// TwinCAT 3 PLC project Nepionic_PackML_Test
// ProgramVersion: 3.1.4026.21
// libraries:
//   [Nepionic_PackML], * (Nepionic)
//   Tc3_Module, * (Beckhoff Automation GmbH)
//   TcUnit, * (www.tcunit.org)
// project tree:
//   Mocks/ MockUnitMode.TcPOU
//   Programs/ TestRunner.TcPOU
//   Tasks/ TestRunnerTask.TcTTO
//   Tests/ PackMLTestSuite.TcPOU
// real-time tasks:
//   TASK TestRunnerTask: cycle T#10ms, priority 20, ADS port 350

CONFIGURATION Nepionic_PackML_Test
    RESOURCE PLC ON TwinCAT3
        TASK TestRunnerTask(INTERVAL := T#10ms, PRIORITY := 20);
        PROGRAM TestRunner WITH TestRunnerTask : TestRunner;
    END_RESOURCE
END_CONFIGURATION

// ---- Programs/TestRunner.TcPOU
PROGRAM TestRunner
VAR
 	packml_test_suite : PackMLTestSuite;
	unit_mode : MockUnitMode;
END_VAR

TcUnit.Run();

END_PROGRAM

// ---- Tests/PackMLTestSuite.TcPOU
FUNCTION_BLOCK PackMLTestSuite EXTENDS TcUnit.FB_TestSuite
VAR
END_VAR

CheckBasicStateMachineCycle();

METHOD PUBLIC CheckBasicStateMachineCycle
VAR_INST
	state_machine : StateMachine<State.Idle>;
END_VAR
Test('CheckStateMachine');

AssertTrue(
	Condition := state_machine.IsIdle,
	Message := 'State machine is not in Idle state immediately after creation'
);

state_machine.Start();
AssertTrue(
	Condition := state_machine.IsStarting,
	Message := 'State machine is not in Starting state immediately after Start action'
);

state_machine.StateComplete();
AssertTrue(
	Condition := state_machine.IsExecuting,
	Message := 'State machine is not in Execute state immediately after Starting state complete'
);

state_machine.StateComplete();
AssertTrue(
	Condition := state_machine.IsCompleting,
	Message := 'State machine is not in Completing state immediately after Execute state complete'
);

state_machine.StateComplete();
AssertTrue(
	Condition := state_machine.IsCompleted,
	Message := 'State machine is not in Completed state immediately after Completing state complete'
);

state_machine.Reset();
AssertTrue(
	Condition := state_machine.IsResetting,
	Message := 'State machine is not in Resetting state immediately after Reset action'
);

state_machine.StateComplete();
AssertTrue(
	Condition := state_machine.IsIdle,
	Message := 'State machine is not in Idle state immediately after Resetting state complete'
);

Test_Finished();
END_METHOD

END_FUNCTION_BLOCK

// ---- Mocks/MockUnitMode.TcPOU
{attribute 'linkalways'} 
{attribute 'no_explicit_call' := 'This FB is a CLASS and must be accessed using methods or properties'}
{attribute 'enable_dynamic_creation'}
FUNCTION_BLOCK MockUnitMode EXTENDS DefaultUnitMode<State.Idle>
VAR
END_VAR

METHOD PUBLIC StateComplete
state_machine.StateComplete();
END_METHOD

END_FUNCTION_BLOCK
